ABB RobotStudio station: Obelix1_20190227-010527.rsstn

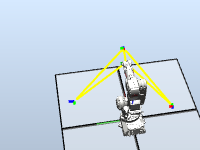
Station Obelix1 (saved by RobotStudio 6.8.8148.134)
Controller IRB_140_6kg_0.81m
  mechanical unit ROB_1: IRB140_6_81_C_03, 6 joints, base frame (0, 0, 0) mm
Layout (positions relative to the parent item):
  - IRB140_6_81_C_03 [mechanism, from Robots\IRB140_6_81_C_G_03.rslib] at (0, 0, 0) mm; joint values [0, 0, 0, 0, 0.5236, 0] (rad or m)
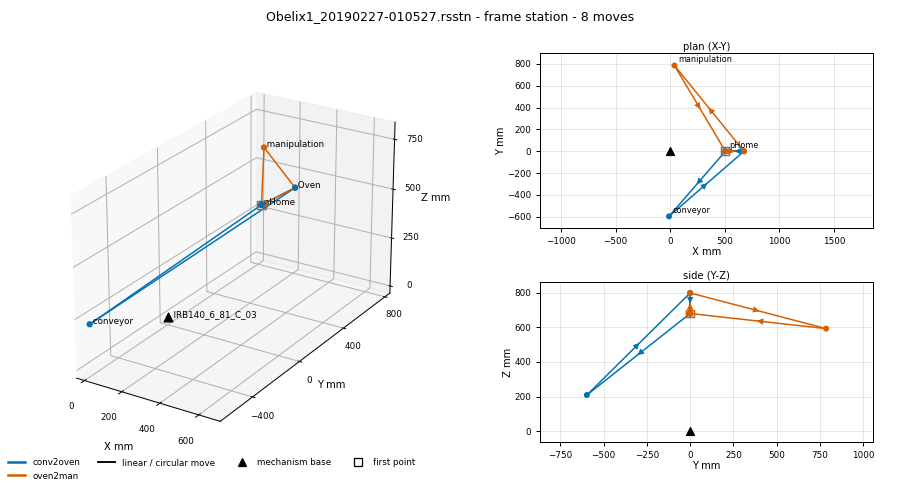
[picture p0: tool path of Obelix1_20190227-010527.rsstn in frame station, 8 of 8 moves have a stored position in this frame; points joined in program order, loops and branches not executed]
Targets, tools, work objects and paths stored in the station, written as RAPID:
! task T_ROB1
MODULE Module1
  CONST robtarget pHome:=[[506.291650772,0,679.49999918],[0.499999994,0,0.866025407,0],[0,0,0,0],[9E+09,9E+09,9E+09,9E+09,9E+09,9E+09]];
  CONST robtarget Oven:=[[676.77830567,0,798.153707831],[0.500000149,0,0.866025318,0],[0,0,0,0],[9E+09,9E+09,9E+09,9E+09,9E+09,9E+09]];
  CONST robtarget conveyor:=[[-9.861164677,-596.337827708,208.8592172],[0.048273193,0.711237174,0.699573246,-0.049078048],[-2,-1,0,0],[9E+09,9E+09,9E+09,9E+09,9E+09,9E+09]];
  CONST robtarget manipulation:=[[40.184227668,785.23645067,592.1503114],[0.554573369,-0.481039839,0.478798532,0.481457181],[0,0,-1,1],[9E+09,9E+09,9E+09,9E+09,9E+09,9E+09]];
  PROC conv2oven()
    MoveL pHome,v1000,z100,tool0\WObj:=wobj0;
    MoveL conveyor,v1000,z100,tool0\WObj:=wobj0;
    MoveL Oven,v1000,z100,tool0\WObj:=wobj0;
    MoveL pHome,v1000,z100,tool0\WObj:=wobj0;
  ENDPROC
  PROC oven2man()
    MoveL pHome,v1000,z100,tool0\WObj:=wobj0;
    MoveL Oven,v1000,z100,tool0\WObj:=wobj0;
    MoveL manipulation,v1000,z100,tool0\WObj:=wobj0;
    MoveL pHome,v1000,z100,tool0\WObj:=wobj0;
  ENDPROC
ENDMODULE

